FUNCTION_BLOCK FB_Stopwatch
VAR_INPUT
	bStart : BOOL;
END_VAR
VAR_OUTPUT
	tElapsed : TIME;
END_VAR
VAR
	stPLC_Task_Info : ST_PLC_TASK_INFORMATION;
	tAccumilator 	: TIME;
	fbTON 			: TON;
END_VAR

IF bStart THEN stPLC_Task_Info := F_Get_PLC_Task_Information(); END_IF
fbTON(PT := stPLC_Task_Info.tCycleTime*2 + tAccumilator);
fbTON(IN := bStart AND NOT(fbTON.Q));
tAccumilator := fbTON.ET; 
IF bStart THEN tElapsed := tAccumilator; END_IF

END_FUNCTION_BLOCK

(* stored: Version 1.1.0.1, ProductVersion 3.1.4024.4
   POU FB_Stopwatch: Id {da9797a0-ade6-4f37-a611-8bc6861938d0}, SpecialFunc None *)
